Universal Robots URScript: timer.script

# timer1: start
# timer2: stop
# timer3: reset

def unnamed():
  global _hidden_verificationVariable=0
  step_count_c2ef86b0_2d39_4edc_9ee2_d099a9e2ee7f = 0.0
  thread Step_Counter_Thread_463eda27_3e90_432b_a9bd_81f2a2cc8606():
    while (True):
      step_count_c2ef86b0_2d39_4edc_9ee2_d099a9e2ee7f = step_count_c2ef86b0_2d39_4edc_9ee2_d099a9e2ee7f + 1.0
      sync()
    end
  end
  run Step_Counter_Thread_463eda27_3e90_432b_a9bd_81f2a2cc8606()
  set_gravity([0.0, 0.0, 9.82])
  set_tcp(p[0.0,0.0,0.0,0.0,0.0,0.0])
  set_safety_mode_transition_hardness(1)
  set_standard_analog_input_domain(0, 1)
  set_standard_analog_input_domain(1, 1)
  set_tool_analog_input_domain(0, 1)
  set_tool_analog_input_domain(1, 1)
  set_analog_outputdomain(0, 0)
  set_analog_outputdomain(1, 0)
  set_input_actions_to_default()
  set_target_payload(1.000000, [0.000000, 0.000000, 0.000000], [0.001539, 0.001539, 0.001539, 0.000000, 0.000000, 0.000000])
  set_tool_communication(False, 115200, 0, 1, 1.5, 3.5)
  set_tool_output_mode(0)
  set_tool_digital_output_mode(0, 1)
  set_tool_digital_output_mode(1, 1)
  set_tool_voltage(0)
  global i_var_1=10
  global timer_1=0
  global timer_2=0
  global timer_3=0
  global timer_3_is_counting=False
  global timer_2_is_counting=False
  global timer_1_is_counting=False
  thread Timer_Thread():
    while (True):
      if (timer_3_is_counting):
        timer_3 = timer_3 + get_steptime()
      end
      if (timer_2_is_counting):
        timer_2 = timer_2 + get_steptime()
      end
      if (timer_1_is_counting):
        timer_1 = timer_1 + get_steptime()
      end
      sync()
    end
  end
  run Timer_Thread()
  while (True):
    $ 1 "Robot Program"
    $ 2 "timer_1: Start"
    timer_1_is_counting = True
    $ 3 "timer_2: Stop"
    timer_2_is_counting = False
    $ 4 "timer_3: Reset"
    timer_3 = 0
  end
end
